_CFC_ (* Continuous Function Chart, elements in execution order *)
#0 OR(SCHU_P2_2_UE2_VL_RESET, SCHU_P2_2_SB)
#1 SEL(UE1_VL_FILTER_ON, T#0ms, T#2s)
#2 fb_UE2_VL:ISTOK_ANALOGVH(enable: TRUE, rawValue: SCHU_P2_2_UE1_AI5, reset: #0, enableLimitCtrl: TRUE, ctrlVoltage: NOT UE1_VL_CVOLT, changeValueWithoutPower: TRUE, highRange: VL_HIGHRANGE, lowRange: VL_LOWRANGE, highLimit: SCHU_P2_2_VL_HIGHLIMIT, lowLimit: SCHU_P2_2_VL_LOWLIMIT, filterTime: #1, offset: ofset, delayEnable: VL_DELAY)
#3 SCHU_P2_2_UE1_VL_VN <= #2.presentValue
#4 SCHU_P2_2_UE1_VL_DOST <= #2.reliability
_END_CFC_
(* the same logic as Structured Text *)
fb_UE2_VL(enable := TRUE, rawValue := SCHU_P2_2_UE1_AI5, reset := SCHU_P2_2_UE2_VL_RESET OR SCHU_P2_2_SB, enableLimitCtrl := TRUE, ctrlVoltage := NOT UE1_VL_CVOLT, changeValueWithoutPower := TRUE, highRange := VL_HIGHRANGE, lowRange := VL_LOWRANGE, highLimit := SCHU_P2_2_VL_HIGHLIMIT, lowLimit := SCHU_P2_2_VL_LOWLIMIT, filterTime := SEL(UE1_VL_FILTER_ON, T#0ms, T#2s), offset := ofset, delayEnable := VL_DELAY);
SCHU_P2_2_UE1_VL_VN := fb_UE2_VL.presentValue;
SCHU_P2_2_UE1_VL_DOST := fb_UE2_VL.reliability;
END_PROGRAM

(* POU TZBiS/TZB/Z_P_PrevDav, CFC *)
PROGRAM Z_P_PrevDav
VAR
	TON_BPrevDav: TON;
	SR_BPerDav: SR;
	TON_PrevDav_P: TON;
END_VAR
VAR (* helpers for the ST form of the networks *)
	_t30 : TIME;
END_VAR
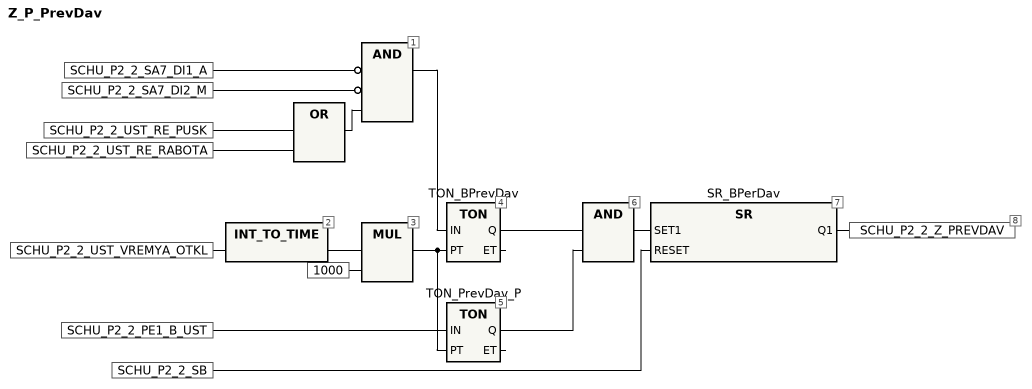
_CFC_ (* Continuous Function Chart, elements in execution order *)
#0 OR(SCHU_P2_2_UST_RE_PUSK, SCHU_P2_2_UST_RE_RABOTA)
#1 AND(NOT SCHU_P2_2_SA7_DI1_A, NOT SCHU_P2_2_SA7_DI2_M, #0)
#2 INT_TO_TIME(SCHU_P2_2_UST_VREMYA_OTKL)
#3 MUL(#2, 1000)
#4 TON_BPrevDav:TON(IN: #1, PT: #3)
#5 TON_PrevDav_P:TON(IN: SCHU_P2_2_PE1_B_UST, PT: #3)
#6 AND(#4.Q, #5.Q)
#7 SR_BPerDav:SR(SET1: #6, RESET: SCHU_P2_2_SB)
#8 SCHU_P2_2_Z_PREVDAV <= #7.Q1
_END_CFC_
(* the same logic as Structured Text *)
_t30 := INT_TO_TIME(SCHU_P2_2_UST_VREMYA_OTKL) * 1000;
TON_BPrevDav(IN := NOT SCHU_P2_2_SA7_DI1_A AND NOT SCHU_P2_2_SA7_DI2_M AND (SCHU_P2_2_UST_RE_PUSK OR SCHU_P2_2_UST_RE_RABOTA), PT := _t30);
TON_PrevDav_P(IN := SCHU_P2_2_PE1_B_UST, PT := _t30);
SR_BPerDav(SET1 := TON_BPrevDav.Q AND TON_PrevDav_P.Q, RESET := SCHU_P2_2_SB);
SCHU_P2_2_Z_PREVDAV := SR_BPerDav.Q1;
END_PROGRAM
